(* CoDeSys 2.3 export: SEQUENTIAL_CTRL.EXP *)

(* POU SEQUENTIAL_CTRL, FBD *)
FUNCTION_BLOCK SEQUENTIAL_CTRL
VAR_INPUT
	xRESET	:	BOOL;
	xT_0_1	:	BOOL;
	xT_1_2	:	BOOL;
	xT_2_3	:	BOOL;
	xT_3_0	:	BOOL;
END_VAR
VAR_OUTPUT
	_xSTEP		:	INT;
END_VAR
VAR
	ctu_step		:	CTU;
END_VAR
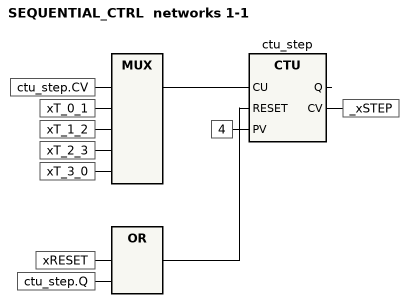
_FBD_ (* Function Block Diagram *)
NETWORK 1
	ctu_step:CTU(CU: MUX(ctu_step.CV, xT_0_1, xT_1_2, xT_2_3, xT_3_0), RESET: OR(xRESET, ctu_step.Q), PV: 4, CV => _xSTEP)
_END_FBD_
(* the same logic as Structured Text *)
(* Network 1 *)
ctu_step(CU := MUX(ctu_step.CV, xT_0_1, xT_1_2, xT_2_3, xT_3_0), RESET := xRESET OR ctu_step.Q, PV := 4);
_xSTEP := ctu_step.CV;
END_FUNCTION_BLOCK
